{attribute 'OPC.UA.DA' := '1'}
{attribute 'OPC.UA.DA.StructuredType' := '1'}
TYPE MaxPowerMsg :
STRUCT
	Id : EPowerIlluminationFlow;
	MaxPower : LREAL;
END_STRUCT
END_TYPE

(* stored: Version 1.1.0.1, ProductVersion 3.1.4024.3
   DUT MaxPowerMsg: Id {6c0f1d23-a724-4f5d-91e7-deaa3f746783} *)
